Yaskawa INFORM job: MOTOMAN.JBI

/JOB
//NAME MOTOMAN
//POS
///NPOS 2,0,0,0,0,0
///TOOL 0
///POSTYPE PULSE
///PULSE
C00000=0,0,0,0,0,0
C00001=107647,26006,0,0,0,0
//INST
///DATE 2009/01/15 17:41
///ATTR RW
///GROUP1 RB1
NOP
MOVJ C00000 VJ=60.00
MOVJ C00001 VJ=60.00
END
